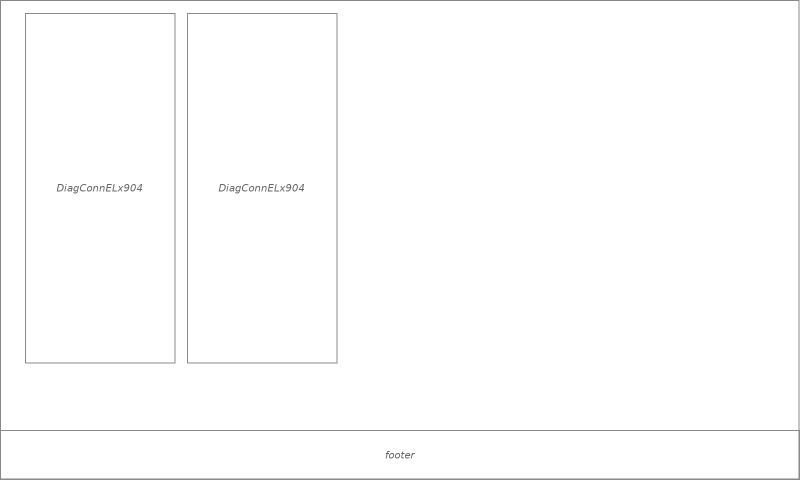
VISUALIZATION ConnDiag  // 800x480
    Frame (0,430 800x50)
        shows footer()
    Frame (25,13 150x350)
        shows DiagConnELx904(connName := 'EL 1904', diag := safetyDiag.diagEL1904, state := safetyDiag.stateEL1904, bits := safetyDiag.el1904Bits)
    Frame (187,13 150x350)
        shows DiagConnELx904(connName := 'EL 2904', diag := safetyDiag.diagEL2904, state := safetyDiag.stateEL2904, bits := safetyDiag.el2904Bits)
END_VISUALIZATION

(* stored: Version 1.1.0.1, ProductVersion 3.1.4024.12
   Visu ConnDiag: Id {f97a6859-ffba-42a7-b14f-7c2682ea481f} *)
